INTERFACE PUBLIC I_Cyclical EXTENDS __System.IQueryInterface

END_INTERFACE

(* stored: Version 1.1.0.1
   Itf I_Cyclical: Id {29724a98-39fb-49ef-8269-a4963832a6e1} *)
